INTERFACE I_QueueDisposedEvent EXTENDS I_Event

PROPERTY PUBLIC TargetQueue : I_Queue
GET
END_GET
END_PROPERTY

END_INTERFACE

(* stored: Version 1.1.0.1, ProductVersion 3.1.4024.12
   Itf I_QueueDisposedEvent: Id {75835e9f-8228-46b3-960f-942c00d6498b}
   Property TargetQueue: Id {97c3064f-c48f-4d86-9fea-0e87873fce6d}
   Get Get: Id {78c9dc8c-e028-4b36-83de-534ee987c836} *)
